FUNCTION Convert_USINT_TO_USINT : Hresult
VAR_INPUT
	in : USINT;
	out : REFERENCE TO USINT;
END_VAR

out := in;

END_FUNCTION

(* stored: Version 1.1.0.1, ProductVersion 3.1.4024.12
   POU Convert_USINT_TO_USINT: Id {e1a5c736-8be1-4628-b126-4e1b90b95e21}, SpecialFunc None *)
